// TIA Portal V16 export
// export: Created 2022-11-17T11:55:29.3196458Z, ExportSetting WithDefaults, DisplayName Totally Integrated Automation Portal, DisplayVersion V16 Update 6, DisplayName TIA Portal Version Control Interface, DisplayVersion V16 Update 2, DisplayName TIA Portal Openness, DisplayVersion V16 Update 6, DisplayName SINAMICS Startdrive Advanced, DisplayVersion V16 Update 5, DisplayName SINAMICS Startdrive G130, G150, S120, S150, SINAMICS MV, S210, DisplayVersion V16 Update 5, DisplayName SINAMICS Startdrive G110M, G120, G120C, G120D, G120P, G115D, DisplayVersion V16 Update 5, DisplayName STEP 7 Professional, DisplayVersion V16 Update 6, DisplayName STEP 7 Safety, DisplayVersion V16, DisplayName WinCC Advanced, DisplayVersion V16 Update 6
DATA_BLOCK "DB26"   // DB26
{ S7_Optimized_Access := 'FALSE' }
VERSION : 0.1
// stored: AutoNumber false, IsOnlyStoredInLoadMemory false, IsWriteProtectedInAS false
   VAR RETAIN
      Dbd0 : Real := 0.0;   // Valore massimo di scalatura dell'uscita = 32000
      Dbd4 : Real := 0.0;   // Valore minimo di scalatura dell'uscita = 0.0
      Dbd8 : Real := 0.0;   // Valore massimo di scalatura della parola di ingresso = 100-%tiro
      Dbd12 : Real := 0.0;   // Valore minimo di scalatura della parola di ingresso analogico = 0.0
      Dbd16 : DInt := 0;   // valore di prestiro impostato sul display convertito a 32 bit
      Dbd20 : Real := 0.0;   // valore di prestiro impostato sul display a 32 bit convertito in virgola mobile
      Dbd24 : Real := 0.0;   // Differenza fra valore massimo di scal.e valore minimo di scal.all'uscita
      Dbd28 : Real := 0.0;   // Differenza fra valore massimo di scal.e valore minimo di scal.all'input analogi
      Dbd32 : Real := 0.0;   // differenza fra dbd20 e dbd 12
      Dbd36 : Real := 0.0;
      Dbd40 : Real := 0.0;
      Dbd44 : Real := 0.0;
      Dbw48 : Int := 0;
      Dbw50 : Int := 200;   // valore di prestiro impostato sul display a 16 bit
      Dbw52 : Int := 0;   // valore di tiro impostato sul display a 16 bit
      Dbd54 : DInt := 0;
      Dbd58 : DInt := 0;
      Dbd62 : Real := 0.0;
      Dbd66 : Real := 0.0;
      Dbd70 : Real := 0.0;
      Dbd74 : Real := 0.0;
      Dbd78 : Real := 0.0;
      Dbd82 : DInt := 0;
      Dbw86 : Int := 0;   // valore di tiro impostato sul display a 16 bit per ciclo taglio
      Dbw88 : Int := 5;   // valore di tiro impostato sul display a 16 bit per ciclo avvolgitura
      Dbw90 : Int := 0;   // valore di tiro impostato sul display a 16 bit per inizio ciclo
      Dbw92 : Int := 0;
      Dbw94 : Int := 0;
      Dbw96 : Int := 0;
      Dbw98 : Int := 0;
      Dbw100 : Int := 0;
      Dbw102 : Int := 0;
      Dbw104 : Int := 0;
      Dbw106 : Int := 0;
      Dbw108 : Int := 0;
      Dbw110 : Int := 0;
      Dbw112 : Int := 0;
      Dbw114 : Int := 0;
      Dbw116 : Int := 0;
   END_VAR
BEGIN
END_DATA_BLOCK
